Staubli VAL3: aioItem.dtx

public bool bActive
public string sID
public string sName
public aio aAio
public bool bEnable
